// TIA Portal V20 export
TYPE "typeEmDataControlNode"
// stored: Namespace Unit1.Em2
   STRUCT
      jrOutPnPLeft : "LER_typePartData";
      jrOutPnPRight : "LER_typePartData";
   END_STRUCT;
END_TYPE
